INTERFACE I_Button_1

PROPERTY IsPressed : BOOL
GET
END_GET
SET
END_SET
END_PROPERTY

END_INTERFACE

(* stored: Version 1.1.0.1, ProductVersion 3.1.4024.15
   Itf I_Button_1: Id {2d44b9f1-f678-4eb3-a494-0040b4c9153d}
   Property IsPressed: Id {3321e75e-3589-402f-9c10-054fedfa66e3}
   Get Get: Id {c735861f-8f7c-4c35-ae3d-a25f345274cb}
   Set Set: Id {c706873a-28c4-48e6-85eb-e4dd12591fc9} *)
